// TIA Portal V17 export
// export: Created 2025-03-05T08:01:40.2934801Z, ExportSetting WithDefaults, DisplayName Totally Integrated Automation Portal, DisplayVersion V17 Update 8, DisplayName TIA Portal Openness, DisplayVersion V17 Update 8, DisplayName TIA Portal Version Control Interface, DisplayVersion V17, DisplayName SINAMICS Startdrive Advanced, DisplayVersion V17 SP2, DisplayName SINAMICS Startdrive G110M, G120, G120C, G120D, G120P, G115D, DisplayVersion V17 SP2, DisplayName SINAMICS Startdrive G130, G150, S120, S150, SINAMICS MV, S210, DisplayVersion V17 SP2, DisplayName STEP 7 Professional, DisplayVersion V17 Update 8, DisplayName SINUMERIK ONE STEP 7 Toolbox, DisplayVersion V17 Update 12, DisplayName SINUMERIK 840D sl STEP 7 Toolbox, DisplayVersion V17 Update 12, DisplayName STEP 7 Safety, DisplayVersion V17 Update 6, DisplayName WinCC Advanced, DisplayVersion V17 Update 8
FUNCTION "FC7222_MACHINE_OVERVIEW_CLADDING" : Void   // FC7222, LAD
{ S7_Optimized_Access := 'FALSE' }
AUTHOR : ETXETAR
VERSION : 1.0
// stored: AutoNumber false, IsIECCheckEnabled false, SetENOAutomatically false, UDAEnableTagReadback false
   VAR_TEMP
      OPTION_OFF : Bool;   // OPTION OFF
      OPTION_ON : Bool;   // OPTION ON
      SPINDLE_SP11 : Bool;   // SPINDLE SP11
      SPINDLE_SP12 : Bool;   // SPINDLE SP12
      SPINDLE_SP13 : Bool;   // SPINDLE SP13
      SPINDLE_SP14 : Bool;   // SPINDLE SP14
      SPINDLE_SP21 : Bool;   // SPINDLE SP21
      SPINDLE_SP22 : Bool;   // SPINDLE SP22
      SPINDLE_SP23 : Bool;   // SPINDLE SP23
      SPINDLE_SP24 : Bool;   // SPINDLE SP24
      MACH_FIXTURE_1 : Bool;   // MACH FIXTURE 1
      MACH_FIXTURE_2 : Bool;   // MACH FIXTURE 2
      UNIT_MODE_AUX : Int;   // UNIT MODE AUXILIARY
   END_VAR
   VAR_TEMP   // added for the SCL form of the ladder/FBD networks
      _w1 : Bool;
      _w2 : Bool;
      _w3 : Bool;
      _w4 : Bool;
   END_VAR
BEGIN

REGION Network 1: OPTION OFF
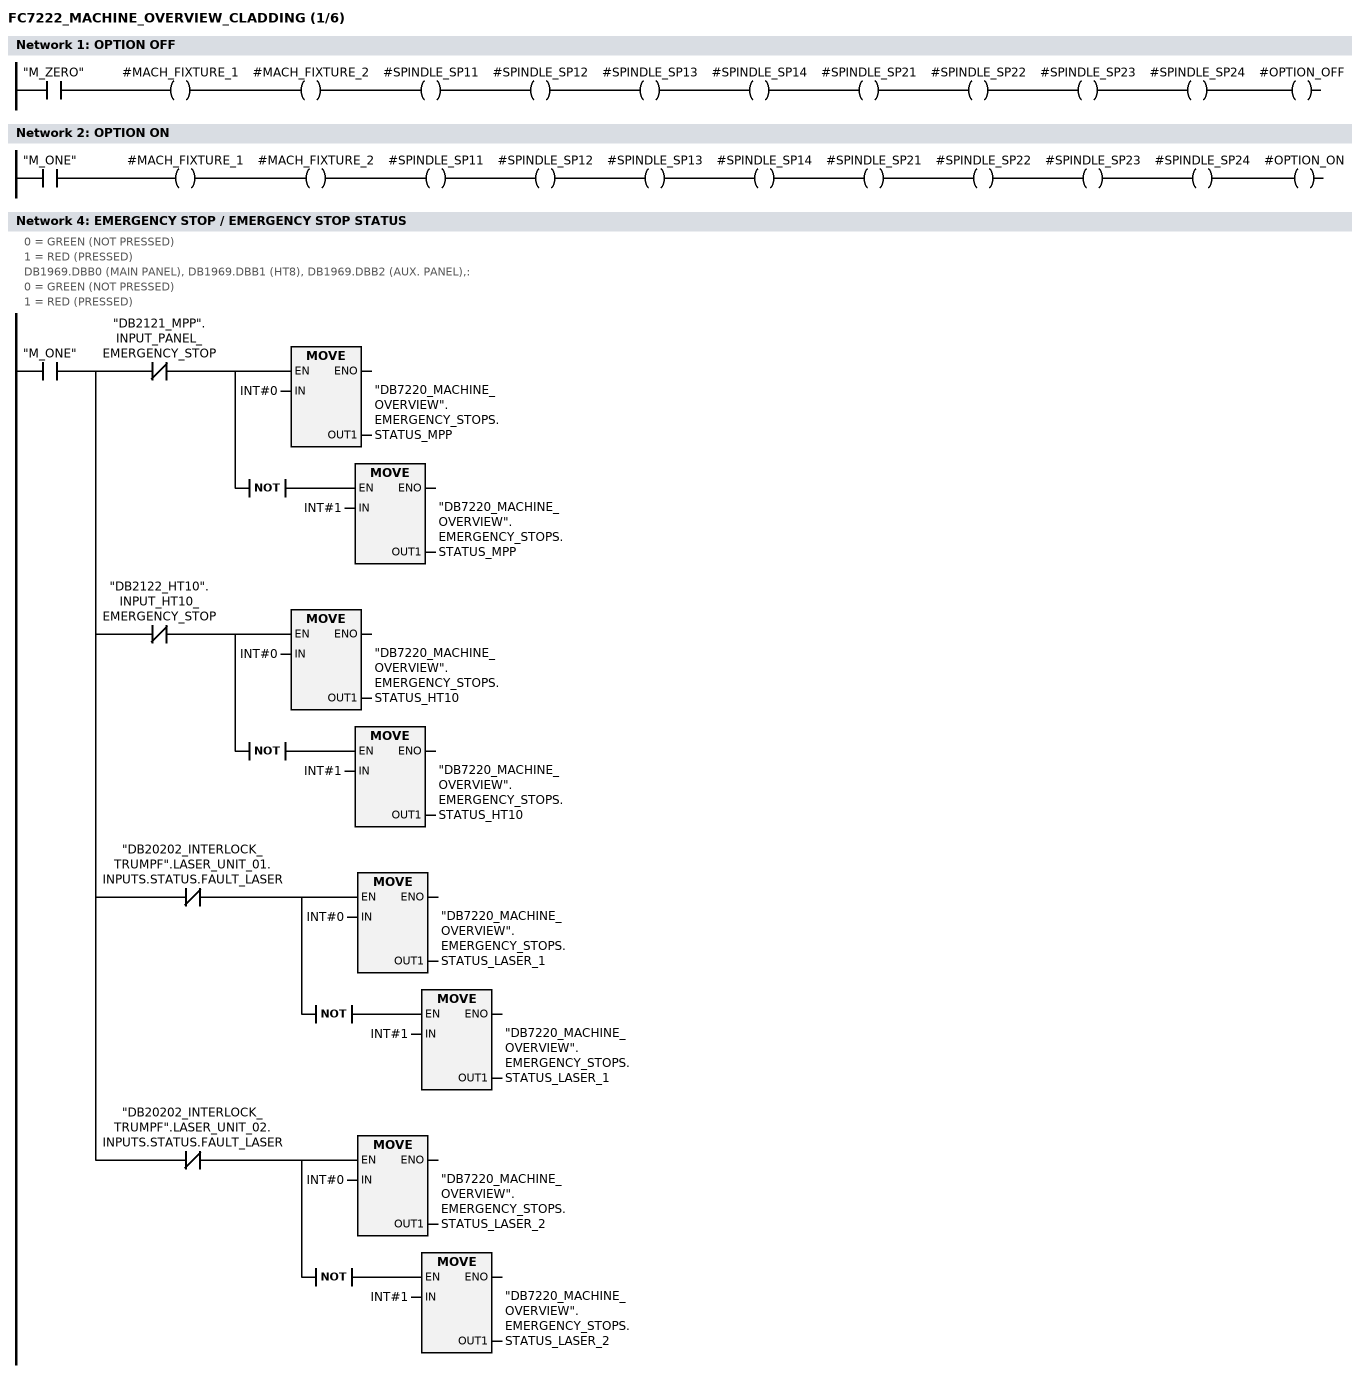
   RUNG wire#powerrail
      Contact( "M_ZERO" )
      Coil( #MACH_FIXTURE_1 )
      Coil( #MACH_FIXTURE_2 )
      Coil( #SPINDLE_SP11 )
      Coil( #SPINDLE_SP12 )
      Coil( #SPINDLE_SP13 )
      Coil( #SPINDLE_SP14 )
      Coil( #SPINDLE_SP21 )
      Coil( #SPINDLE_SP22 )
      Coil( #SPINDLE_SP23 )
      Coil( #SPINDLE_SP24 )
      Coil( #OPTION_OFF )
   END_RUNG
   // the same network as SCL:
   #MACH_FIXTURE_1 := "M_ZERO";
   #MACH_FIXTURE_2 := "M_ZERO";
   #SPINDLE_SP11 := "M_ZERO";
   #SPINDLE_SP12 := "M_ZERO";
   #SPINDLE_SP13 := "M_ZERO";
   #SPINDLE_SP14 := "M_ZERO";
   #SPINDLE_SP21 := "M_ZERO";
   #SPINDLE_SP22 := "M_ZERO";
   #SPINDLE_SP23 := "M_ZERO";
   #SPINDLE_SP24 := "M_ZERO";
   #OPTION_OFF := "M_ZERO";
END_REGION

REGION Network 2: OPTION ON
   RUNG wire#powerrail
      Contact( "M_ONE" )
      Coil( #MACH_FIXTURE_1 )
      Coil( #MACH_FIXTURE_2 )
      Coil( #SPINDLE_SP11 )
      Coil( #SPINDLE_SP12 )
      Coil( #SPINDLE_SP13 )
      Coil( #SPINDLE_SP14 )
      Coil( #SPINDLE_SP21 )
      Coil( #SPINDLE_SP22 )
      Coil( #SPINDLE_SP23 )
      Coil( #SPINDLE_SP24 )
      Coil( #OPTION_ON )
   END_RUNG
   // the same network as SCL:
   #MACH_FIXTURE_1 := "M_ONE";
   #MACH_FIXTURE_2 := "M_ONE";
   #SPINDLE_SP11 := "M_ONE";
   #SPINDLE_SP12 := "M_ONE";
   #SPINDLE_SP13 := "M_ONE";
   #SPINDLE_SP14 := "M_ONE";
   #SPINDLE_SP21 := "M_ONE";
   #SPINDLE_SP22 := "M_ONE";
   #SPINDLE_SP23 := "M_ONE";
   #SPINDLE_SP24 := "M_ONE";
   #OPTION_ON := "M_ONE";
END_REGION

REGION Network 3: ********** EMERGENCY STOP **********
   // MPP PANEL EMERGENCY STOP
   // HT10 EMERGENCY STOP
   // AUXILIAR MAGAZINE PANEL EMERGENCY STOP
   // MANUAL LOADING EMERGENCY STOP
   // CHIP CONVEYOR EMERGENCY STOP
END_REGION

REGION Network 4: EMERGENCY STOP / EMERGENCY STOP STATUS
   // 0 = GREEN (NOT PRESSED)
   // 1 = RED (PRESSED)
   // DB1969.DBB0 (MAIN PANEL), DB1969.DBB1 (HT8), DB1969.DBB2 (AUX. PANEL),:
   // 
   // 0 = GREEN (NOT PRESSED)
   // 
   // 1 = RED (PRESSED)
   RUNG wire#powerrail
      Contact( "M_ONE" )
      wire#w1
      I_Contact( "DB2121_MPP".INPUT_PANEL_EMERGENCY_STOP )
      wire#w2
      { S7_GenerateENO := "TRUE" } Move(in := INT#0, out1 => "DB7220_MACHINE_OVERVIEW".EMERGENCY_STOPS.STATUS_MPP)
   END_RUNG
   RUNG wire#w2
      Not()
      { S7_GenerateENO := "TRUE" } Move(in := INT#1, out1 => "DB7220_MACHINE_OVERVIEW".EMERGENCY_STOPS.STATUS_MPP)
   END_RUNG
   RUNG wire#w1
      I_Contact( "DB2122_HT10".INPUT_HT10_EMERGENCY_STOP )
      wire#w3
      { S7_GenerateENO := "TRUE" } Move(in := INT#0, out1 => "DB7220_MACHINE_OVERVIEW".EMERGENCY_STOPS.STATUS_HT10)
   END_RUNG
   RUNG wire#w3
      Not()
      { S7_GenerateENO := "TRUE" } Move(in := INT#1, out1 => "DB7220_MACHINE_OVERVIEW".EMERGENCY_STOPS.STATUS_HT10)
   END_RUNG
   RUNG wire#w1
      I_Contact( "DB20202_INTERLOCK_TRUMPF".LASER_UNIT_01.INPUTS.STATUS.FAULT_LASER )
      wire#w4
      Move(in := INT#0, out1 => "DB7220_MACHINE_OVERVIEW".EMERGENCY_STOPS.STATUS_LASER_1)
   END_RUNG
   RUNG wire#w4
      Not()
      Move(in := INT#1, out1 => "DB7220_MACHINE_OVERVIEW".EMERGENCY_STOPS.STATUS_LASER_1)
   END_RUNG
   RUNG wire#w1
      I_Contact( "DB20202_INTERLOCK_TRUMPF".LASER_UNIT_02.INPUTS.STATUS.FAULT_LASER )
      wire#w5
      Move(in := INT#0, out1 => "DB7220_MACHINE_OVERVIEW".EMERGENCY_STOPS.STATUS_LASER_2)
   END_RUNG
   RUNG wire#w5
      Not()
      Move(in := INT#1, out1 => "DB7220_MACHINE_OVERVIEW".EMERGENCY_STOPS.STATUS_LASER_2)
   END_RUNG
   // the same network as SCL:
   #_w1 := "M_ONE" AND NOT "DB2121_MPP".INPUT_PANEL_EMERGENCY_STOP;
   IF #_w1 THEN "DB7220_MACHINE_OVERVIEW".EMERGENCY_STOPS.STATUS_MPP := INT#0; END_IF;
   IF NOT #_w1 THEN "DB7220_MACHINE_OVERVIEW".EMERGENCY_STOPS.STATUS_MPP := INT#1; END_IF;
   #_w2 := "M_ONE" AND NOT "DB2122_HT10".INPUT_HT10_EMERGENCY_STOP;
   IF #_w2 THEN "DB7220_MACHINE_OVERVIEW".EMERGENCY_STOPS.STATUS_HT10 := INT#0; END_IF;
   IF NOT #_w2 THEN "DB7220_MACHINE_OVERVIEW".EMERGENCY_STOPS.STATUS_HT10 := INT#1; END_IF;
   #_w3 := "M_ONE" AND NOT "DB20202_INTERLOCK_TRUMPF".LASER_UNIT_01.INPUTS.STATUS.FAULT_LASER;
   IF #_w3 THEN "DB7220_MACHINE_OVERVIEW".EMERGENCY_STOPS.STATUS_LASER_1 := INT#0; END_IF;
   IF NOT #_w3 THEN "DB7220_MACHINE_OVERVIEW".EMERGENCY_STOPS.STATUS_LASER_1 := INT#1; END_IF;
   #_w4 := "M_ONE" AND NOT "DB20202_INTERLOCK_TRUMPF".LASER_UNIT_02.INPUTS.STATUS.FAULT_LASER;
   IF #_w4 THEN "DB7220_MACHINE_OVERVIEW".EMERGENCY_STOPS.STATUS_LASER_2 := INT#0; END_IF;
   IF NOT #_w4 THEN "DB7220_MACHINE_OVERVIEW".EMERGENCY_STOPS.STATUS_LASER_2 := INT#1; END_IF;
END_REGION

REGION Network 5: ********** SAFETY DOORS **********
   // ::::::::::::::::::::::::::::::::::::::::::::::::::::::::::::::::::::::::::::::::
   // :::::::::::::::::::::::::::: SAFETY DOOR STATUS ::::::::::::::::::::::::::::::::
   // ::::::::::::::::::::::::::::::::::::::::::::::::::::::::::::::::::::::::::::::::
   // DELETE THE NETWORKS OF THE DOORS THAT DO NOT EXIST IN THE MACHINE
   // TOOL MAGAZINE 01R SAFETY DOOR
   // TOOL MAGAZINE 01L SAFETY DOOR
   // UNIT 01R SAFETY DOOR
   // UNIT 01L SAFETY DOOR
   // CHIP CONVEYOR SAFETY DOOR
   // AUTOMATIC DOOR
END_REGION

REGION Network 6: UNIT 01 MAIN SAFETY DOOR
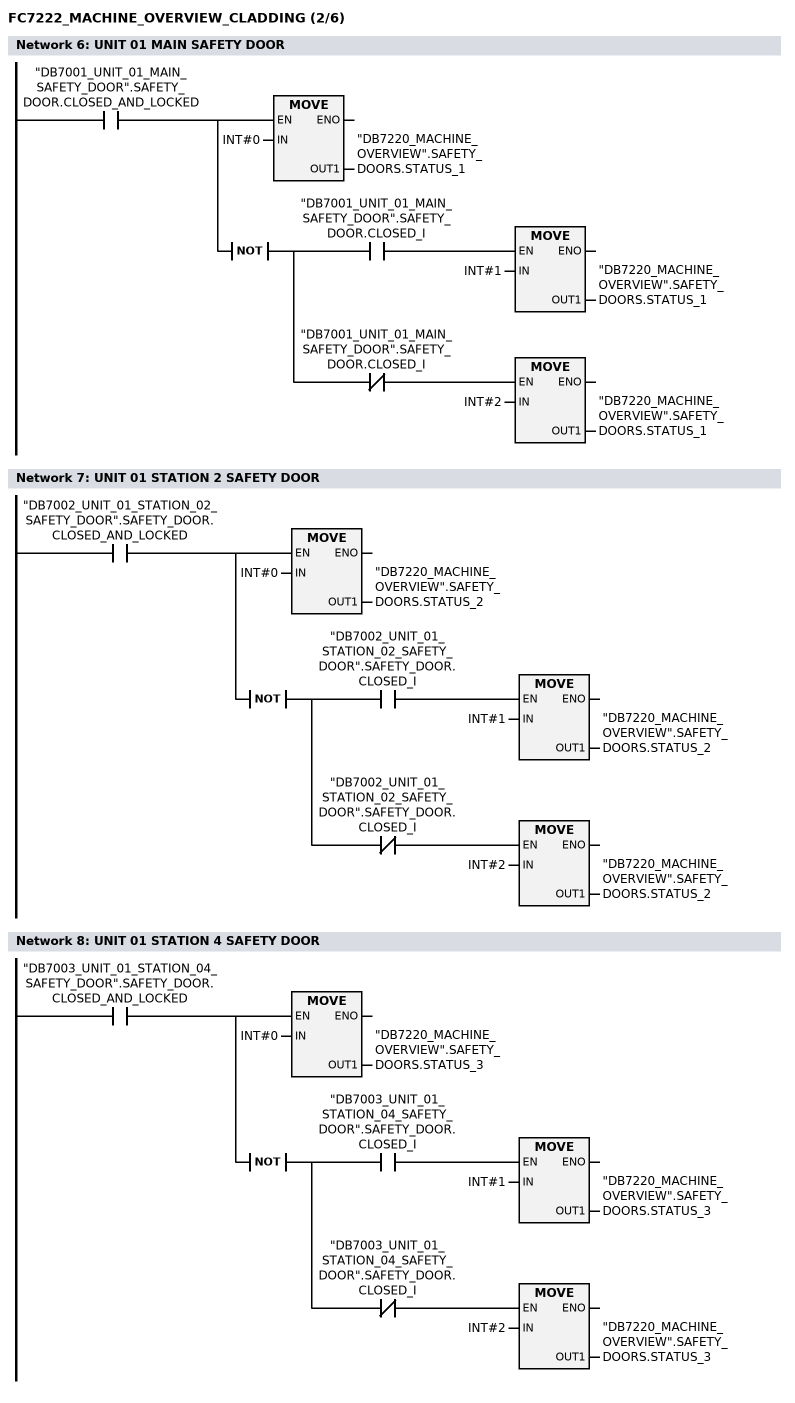
   RUNG wire#powerrail
      Contact( "DB7001_UNIT_01_MAIN_SAFETY_DOOR".SAFETY_DOOR.CLOSED_AND_LOCKED )
      wire#w1
      Move(in := INT#0, out1 => "DB7220_MACHINE_OVERVIEW".SAFETY_DOORS.STATUS_1)
   END_RUNG
   RUNG wire#w1
      Not()
      wire#w2
      Contact( "DB7001_UNIT_01_MAIN_SAFETY_DOOR".SAFETY_DOOR.CLOSED_I )
      Move(in := INT#1, out1 => "DB7220_MACHINE_OVERVIEW".SAFETY_DOORS.STATUS_1)
   END_RUNG
   RUNG wire#w2
      I_Contact( "DB7001_UNIT_01_MAIN_SAFETY_DOOR".SAFETY_DOOR.CLOSED_I )
      Move(in := INT#2, out1 => "DB7220_MACHINE_OVERVIEW".SAFETY_DOORS.STATUS_1)
   END_RUNG
   // the same network as SCL:
   IF "DB7001_UNIT_01_MAIN_SAFETY_DOOR".SAFETY_DOOR.CLOSED_AND_LOCKED THEN
       "DB7220_MACHINE_OVERVIEW".SAFETY_DOORS.STATUS_1 := INT#0;
   END_IF;
   #_w1 := NOT "DB7001_UNIT_01_MAIN_SAFETY_DOOR".SAFETY_DOOR.CLOSED_AND_LOCKED;
   IF #_w1 AND "DB7001_UNIT_01_MAIN_SAFETY_DOOR".SAFETY_DOOR.CLOSED_I THEN
       "DB7220_MACHINE_OVERVIEW".SAFETY_DOORS.STATUS_1 := INT#1;
   END_IF;
   IF #_w1 AND NOT "DB7001_UNIT_01_MAIN_SAFETY_DOOR".SAFETY_DOOR.CLOSED_I THEN
       "DB7220_MACHINE_OVERVIEW".SAFETY_DOORS.STATUS_1 := INT#2;
   END_IF;
END_REGION

REGION Network 7: UNIT 01 STATION 2 SAFETY DOOR
   RUNG wire#powerrail
      Contact( "DB7002_UNIT_01_STATION_02_SAFETY_DOOR".SAFETY_DOOR.CLOSED_AND_LOCKED )
      wire#w1
      Move(in := INT#0, out1 => "DB7220_MACHINE_OVERVIEW".SAFETY_DOORS.STATUS_2)
   END_RUNG
   RUNG wire#w1
      Not()
      wire#w2
      Contact( "DB7002_UNIT_01_STATION_02_SAFETY_DOOR".SAFETY_DOOR.CLOSED_I )
      Move(in := INT#1, out1 => "DB7220_MACHINE_OVERVIEW".SAFETY_DOORS.STATUS_2)
   END_RUNG
   RUNG wire#w2
      I_Contact( "DB7002_UNIT_01_STATION_02_SAFETY_DOOR".SAFETY_DOOR.CLOSED_I )
      Move(in := INT#2, out1 => "DB7220_MACHINE_OVERVIEW".SAFETY_DOORS.STATUS_2)
   END_RUNG
   // the same network as SCL:
   IF "DB7002_UNIT_01_STATION_02_SAFETY_DOOR".SAFETY_DOOR.CLOSED_AND_LOCKED THEN
       "DB7220_MACHINE_OVERVIEW".SAFETY_DOORS.STATUS_2 := INT#0;
   END_IF;
   #_w1 := NOT "DB7002_UNIT_01_STATION_02_SAFETY_DOOR".SAFETY_DOOR.CLOSED_AND_LOCKED;
   IF #_w1 AND "DB7002_UNIT_01_STATION_02_SAFETY_DOOR".SAFETY_DOOR.CLOSED_I THEN
       "DB7220_MACHINE_OVERVIEW".SAFETY_DOORS.STATUS_2 := INT#1;
   END_IF;
   IF #_w1 AND NOT "DB7002_UNIT_01_STATION_02_SAFETY_DOOR".SAFETY_DOOR.CLOSED_I THEN
       "DB7220_MACHINE_OVERVIEW".SAFETY_DOORS.STATUS_2 := INT#2;
   END_IF;
END_REGION

REGION Network 8: UNIT 01 STATION 4 SAFETY DOOR
   RUNG wire#powerrail
      Contact( "DB7003_UNIT_01_STATION_04_SAFETY_DOOR".SAFETY_DOOR.CLOSED_AND_LOCKED )
      wire#w1
      Move(in := INT#0, out1 => "DB7220_MACHINE_OVERVIEW".SAFETY_DOORS.STATUS_3)
   END_RUNG
   RUNG wire#w1
      Not()
      wire#w2
      Contact( "DB7003_UNIT_01_STATION_04_SAFETY_DOOR".SAFETY_DOOR.CLOSED_I )
      Move(in := INT#1, out1 => "DB7220_MACHINE_OVERVIEW".SAFETY_DOORS.STATUS_3)
   END_RUNG
   RUNG wire#w2
      I_Contact( "DB7003_UNIT_01_STATION_04_SAFETY_DOOR".SAFETY_DOOR.CLOSED_I )
      Move(in := INT#2, out1 => "DB7220_MACHINE_OVERVIEW".SAFETY_DOORS.STATUS_3)
   END_RUNG
   // the same network as SCL:
   IF "DB7003_UNIT_01_STATION_04_SAFETY_DOOR".SAFETY_DOOR.CLOSED_AND_LOCKED THEN
       "DB7220_MACHINE_OVERVIEW".SAFETY_DOORS.STATUS_3 := INT#0;
   END_IF;
   #_w1 := NOT "DB7003_UNIT_01_STATION_04_SAFETY_DOOR".SAFETY_DOOR.CLOSED_AND_LOCKED;
   IF #_w1 AND "DB7003_UNIT_01_STATION_04_SAFETY_DOOR".SAFETY_DOOR.CLOSED_I THEN
       "DB7220_MACHINE_OVERVIEW".SAFETY_DOORS.STATUS_3 := INT#1;
   END_IF;
   IF #_w1 AND NOT "DB7003_UNIT_01_STATION_04_SAFETY_DOOR".SAFETY_DOOR.CLOSED_I THEN
       "DB7220_MACHINE_OVERVIEW".SAFETY_DOORS.STATUS_3 := INT#2;
   END_IF;
END_REGION

REGION Network 9: UNIT 02 MAIN SAFETY DOOR
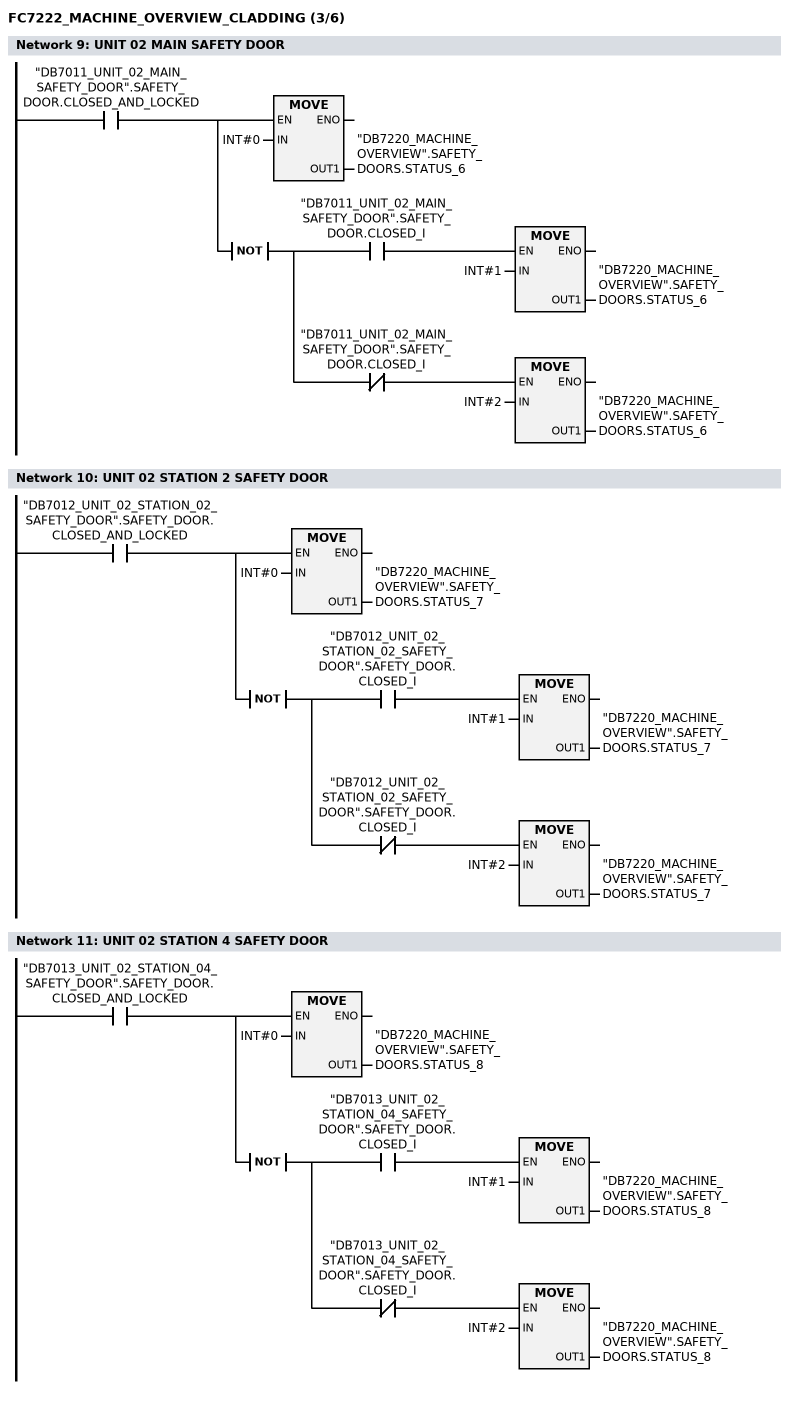
   RUNG wire#powerrail
      Contact( "DB7011_UNIT_02_MAIN_SAFETY_DOOR".SAFETY_DOOR.CLOSED_AND_LOCKED )
      wire#w1
      Move(in := INT#0, out1 => "DB7220_MACHINE_OVERVIEW".SAFETY_DOORS.STATUS_6)
   END_RUNG
   RUNG wire#w1
      Not()
      wire#w2
      Contact( "DB7011_UNIT_02_MAIN_SAFETY_DOOR".SAFETY_DOOR.CLOSED_I )
      Move(in := INT#1, out1 => "DB7220_MACHINE_OVERVIEW".SAFETY_DOORS.STATUS_6)
   END_RUNG
   RUNG wire#w2
      I_Contact( "DB7011_UNIT_02_MAIN_SAFETY_DOOR".SAFETY_DOOR.CLOSED_I )
      Move(in := INT#2, out1 => "DB7220_MACHINE_OVERVIEW".SAFETY_DOORS.STATUS_6)
   END_RUNG
   // the same network as SCL:
   IF "DB7011_UNIT_02_MAIN_SAFETY_DOOR".SAFETY_DOOR.CLOSED_AND_LOCKED THEN
       "DB7220_MACHINE_OVERVIEW".SAFETY_DOORS.STATUS_6 := INT#0;
   END_IF;
   #_w1 := NOT "DB7011_UNIT_02_MAIN_SAFETY_DOOR".SAFETY_DOOR.CLOSED_AND_LOCKED;
   IF #_w1 AND "DB7011_UNIT_02_MAIN_SAFETY_DOOR".SAFETY_DOOR.CLOSED_I THEN
       "DB7220_MACHINE_OVERVIEW".SAFETY_DOORS.STATUS_6 := INT#1;
   END_IF;
   IF #_w1 AND NOT "DB7011_UNIT_02_MAIN_SAFETY_DOOR".SAFETY_DOOR.CLOSED_I THEN
       "DB7220_MACHINE_OVERVIEW".SAFETY_DOORS.STATUS_6 := INT#2;
   END_IF;
END_REGION

REGION Network 10: UNIT 02 STATION 2 SAFETY DOOR
   RUNG wire#powerrail
      Contact( "DB7012_UNIT_02_STATION_02_SAFETY_DOOR".SAFETY_DOOR.CLOSED_AND_LOCKED )
      wire#w1
      Move(in := INT#0, out1 => "DB7220_MACHINE_OVERVIEW".SAFETY_DOORS.STATUS_7)
   END_RUNG
   RUNG wire#w1
      Not()
      wire#w2
      Contact( "DB7012_UNIT_02_STATION_02_SAFETY_DOOR".SAFETY_DOOR.CLOSED_I )
      Move(in := INT#1, out1 => "DB7220_MACHINE_OVERVIEW".SAFETY_DOORS.STATUS_7)
   END_RUNG
   RUNG wire#w2
      I_Contact( "DB7012_UNIT_02_STATION_02_SAFETY_DOOR".SAFETY_DOOR.CLOSED_I )
      Move(in := INT#2, out1 => "DB7220_MACHINE_OVERVIEW".SAFETY_DOORS.STATUS_7)
   END_RUNG
   // the same network as SCL:
   IF "DB7012_UNIT_02_STATION_02_SAFETY_DOOR".SAFETY_DOOR.CLOSED_AND_LOCKED THEN
       "DB7220_MACHINE_OVERVIEW".SAFETY_DOORS.STATUS_7 := INT#0;
   END_IF;
   #_w1 := NOT "DB7012_UNIT_02_STATION_02_SAFETY_DOOR".SAFETY_DOOR.CLOSED_AND_LOCKED;
   IF #_w1 AND "DB7012_UNIT_02_STATION_02_SAFETY_DOOR".SAFETY_DOOR.CLOSED_I THEN
       "DB7220_MACHINE_OVERVIEW".SAFETY_DOORS.STATUS_7 := INT#1;
   END_IF;
   IF #_w1 AND NOT "DB7012_UNIT_02_STATION_02_SAFETY_DOOR".SAFETY_DOOR.CLOSED_I THEN
       "DB7220_MACHINE_OVERVIEW".SAFETY_DOORS.STATUS_7 := INT#2;
   END_IF;
END_REGION

REGION Network 11: UNIT 02 STATION 4 SAFETY DOOR
   RUNG wire#powerrail
      Contact( "DB7013_UNIT_02_STATION_04_SAFETY_DOOR".SAFETY_DOOR.CLOSED_AND_LOCKED )
      wire#w1
      Move(in := INT#0, out1 => "DB7220_MACHINE_OVERVIEW".SAFETY_DOORS.STATUS_8)
   END_RUNG
   RUNG wire#w1
      Not()
      wire#w2
      Contact( "DB7013_UNIT_02_STATION_04_SAFETY_DOOR".SAFETY_DOOR.CLOSED_I )
      Move(in := INT#1, out1 => "DB7220_MACHINE_OVERVIEW".SAFETY_DOORS.STATUS_8)
   END_RUNG
   RUNG wire#w2
      I_Contact( "DB7013_UNIT_02_STATION_04_SAFETY_DOOR".SAFETY_DOOR.CLOSED_I )
      Move(in := INT#2, out1 => "DB7220_MACHINE_OVERVIEW".SAFETY_DOORS.STATUS_8)
   END_RUNG
   // the same network as SCL:
   IF "DB7013_UNIT_02_STATION_04_SAFETY_DOOR".SAFETY_DOOR.CLOSED_AND_LOCKED THEN
       "DB7220_MACHINE_OVERVIEW".SAFETY_DOORS.STATUS_8 := INT#0;
   END_IF;
   #_w1 := NOT "DB7013_UNIT_02_STATION_04_SAFETY_DOOR".SAFETY_DOOR.CLOSED_AND_LOCKED;
   IF #_w1 AND "DB7013_UNIT_02_STATION_04_SAFETY_DOOR".SAFETY_DOOR.CLOSED_I THEN
       "DB7220_MACHINE_OVERVIEW".SAFETY_DOORS.STATUS_8 := INT#1;
   END_IF;
   IF #_w1 AND NOT "DB7013_UNIT_02_STATION_04_SAFETY_DOOR".SAFETY_DOOR.CLOSED_I THEN
       "DB7220_MACHINE_OVERVIEW".SAFETY_DOORS.STATUS_8 := INT#2;
   END_IF;
END_REGION

REGION Network 12: ********** UNITS **********
END_REGION

REGION Network 13: UNIT MODE STATUS
   // 0 = GREEN (AUTO)
   // 
   // 1 = BLUE (MANUAL)
   // 
   // 2 = YELLOW (MDA) 
   // 
   // 3 = WHITE (SEMIAUTOMATIC)
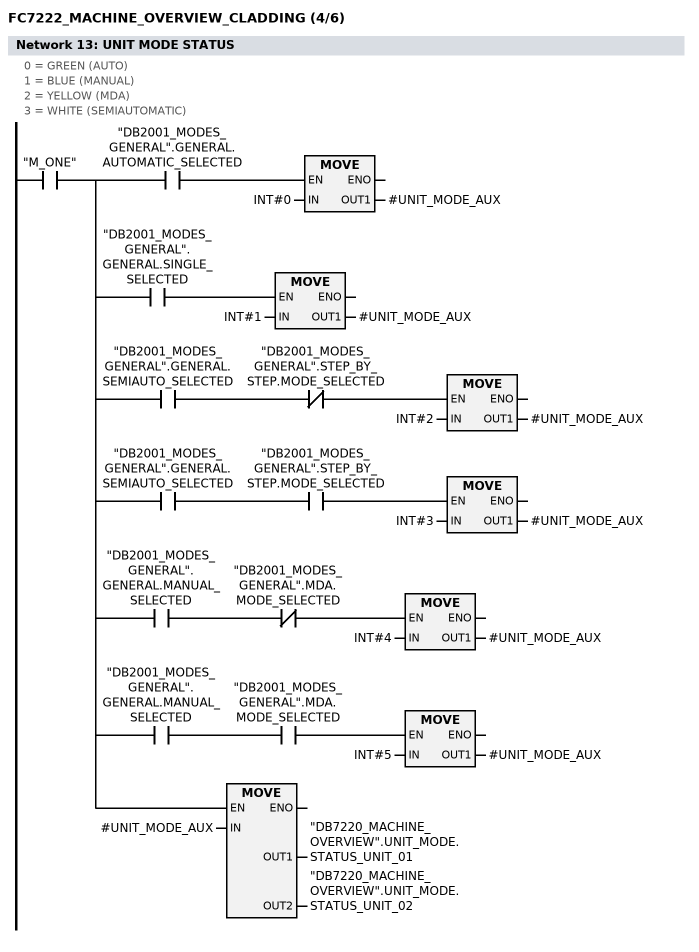
   RUNG wire#powerrail
      Contact( "M_ONE" )
      wire#w1
      Contact( "DB2001_MODES_GENERAL".GENERAL.AUTOMATIC_SELECTED )
      { S7_GenerateENO := "TRUE" } Move(in := INT#0, out1 => #UNIT_MODE_AUX)
   END_RUNG
   RUNG wire#w1
      Contact( "DB2001_MODES_GENERAL".GENERAL.SINGLE_SELECTED )
      { S7_GenerateENO := "TRUE" } Move(in := INT#1, out1 => #UNIT_MODE_AUX)
   END_RUNG
   RUNG wire#w1
      Contact( "DB2001_MODES_GENERAL".GENERAL.SEMIAUTO_SELECTED )
      I_Contact( "DB2001_MODES_GENERAL".STEP_BY_STEP.MODE_SELECTED )
      { S7_GenerateENO := "TRUE" } Move(in := INT#2, out1 => #UNIT_MODE_AUX)
   END_RUNG
   RUNG wire#w1
      Contact( "DB2001_MODES_GENERAL".GENERAL.SEMIAUTO_SELECTED )
      Contact( "DB2001_MODES_GENERAL".STEP_BY_STEP.MODE_SELECTED )
      { S7_GenerateENO := "TRUE" } Move(in := INT#3, out1 => #UNIT_MODE_AUX)
   END_RUNG
   RUNG wire#w1
      Contact( "DB2001_MODES_GENERAL".GENERAL.MANUAL_SELECTED )
      I_Contact( "DB2001_MODES_GENERAL".MDA.MODE_SELECTED )
      { S7_GenerateENO := "TRUE" } Move(in := INT#4, out1 => #UNIT_MODE_AUX)
   END_RUNG
   RUNG wire#w1
      Contact( "DB2001_MODES_GENERAL".GENERAL.MANUAL_SELECTED )
      Contact( "DB2001_MODES_GENERAL".MDA.MODE_SELECTED )
      { S7_GenerateENO := "TRUE" } Move(in := INT#5, out1 => #UNIT_MODE_AUX)
   END_RUNG
   RUNG wire#w1
      { S7_GenerateENO := "TRUE" } Move(in := #UNIT_MODE_AUX, out1 => "DB7220_MACHINE_OVERVIEW".UNIT_MODE.STATUS_UNIT_01, out2 => "DB7220_MACHINE_OVERVIEW".UNIT_MODE.STATUS_UNIT_02)
   END_RUNG
   // the same network as SCL:
   IF "M_ONE" AND "DB2001_MODES_GENERAL".GENERAL.AUTOMATIC_SELECTED THEN #UNIT_MODE_AUX := INT#0; END_IF;
   IF "M_ONE" AND "DB2001_MODES_GENERAL".GENERAL.SINGLE_SELECTED THEN #UNIT_MODE_AUX := INT#1; END_IF;
   IF "M_ONE" AND "DB2001_MODES_GENERAL".GENERAL.SEMIAUTO_SELECTED AND NOT "DB2001_MODES_GENERAL".STEP_BY_STEP.MODE_SELECTED THEN
       #UNIT_MODE_AUX := INT#2;
   END_IF;
   IF "M_ONE" AND "DB2001_MODES_GENERAL".GENERAL.SEMIAUTO_SELECTED AND "DB2001_MODES_GENERAL".STEP_BY_STEP.MODE_SELECTED THEN
       #UNIT_MODE_AUX := INT#3;
   END_IF;
   IF "M_ONE" AND "DB2001_MODES_GENERAL".GENERAL.MANUAL_SELECTED AND NOT "DB2001_MODES_GENERAL".MDA.MODE_SELECTED THEN
       #UNIT_MODE_AUX := INT#4;
   END_IF;
   IF "M_ONE" AND "DB2001_MODES_GENERAL".GENERAL.MANUAL_SELECTED AND "DB2001_MODES_GENERAL".MDA.MODE_SELECTED THEN
       #UNIT_MODE_AUX := INT#5;
   END_IF;
   IF "M_ONE" THEN
       "DB7220_MACHINE_OVERVIEW".UNIT_MODE.STATUS_UNIT_01 := #UNIT_MODE_AUX;
       "DB7220_MACHINE_OVERVIEW".UNIT_MODE.STATUS_UNIT_02 := #UNIT_MODE_AUX;
   END_IF;
END_REGION

REGION Network 14: UNITS STATUS / MACHINE STATUS UNIT 01R FIELD (UNIT)
   // 0 = GREEN (CYCLE ON)
   // 
   // 1 = YELLOW (WARNING)
   // 
   // 2 = RED    (ALARM)
   // DB1969.DBB60: UNIT 01R
   // 
   // 0 = GREEN (CYCLE ON)
   // 
   // 1 = YELLOW (WARNING)
   // 
   // 2 = RED    (ALARM)
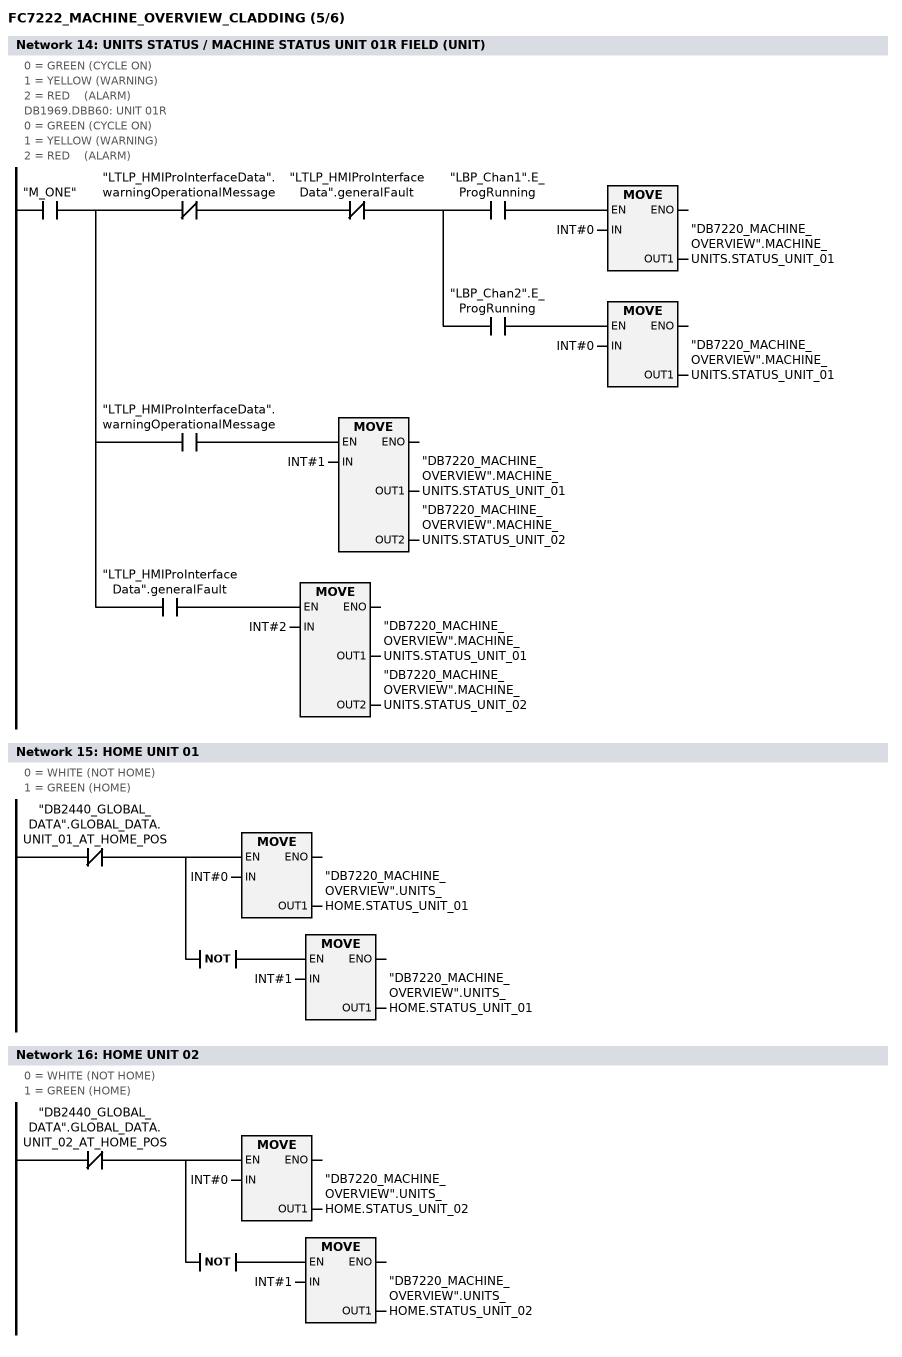
   RUNG wire#powerrail
      Contact( "M_ONE" )
      wire#w1
      I_Contact( "LTLP_HMIProInterfaceData".warningOperationalMessage )
      I_Contact( "LTLP_HMIProInterfaceData".generalFault )
      wire#w2
      Contact( "LBP_Chan1".E_ProgRunning )
      { S7_GenerateENO := "TRUE" } Move(in := INT#0, out1 => "DB7220_MACHINE_OVERVIEW".MACHINE_UNITS.STATUS_UNIT_01)
   END_RUNG
   RUNG wire#w2
      Contact( "LBP_Chan2".E_ProgRunning )
      { S7_GenerateENO := "TRUE" } Move(in := INT#0, out1 => "DB7220_MACHINE_OVERVIEW".MACHINE_UNITS.STATUS_UNIT_01)
   END_RUNG
   RUNG wire#w1
      Contact( "LTLP_HMIProInterfaceData".warningOperationalMessage )
      { S7_GenerateENO := "TRUE" } Move(in := INT#1, out1 => "DB7220_MACHINE_OVERVIEW".MACHINE_UNITS.STATUS_UNIT_01, out2 => "DB7220_MACHINE_OVERVIEW".MACHINE_UNITS.STATUS_UNIT_02)
   END_RUNG
   RUNG wire#w1
      Contact( "LTLP_HMIProInterfaceData".generalFault )
      { S7_GenerateENO := "TRUE" } Move(in := INT#2, out1 => "DB7220_MACHINE_OVERVIEW".MACHINE_UNITS.STATUS_UNIT_01, out2 => "DB7220_MACHINE_OVERVIEW".MACHINE_UNITS.STATUS_UNIT_02)
   END_RUNG
   // the same network as SCL:
   #_w1 := "M_ONE" AND NOT "LTLP_HMIProInterfaceData".warningOperationalMessage AND NOT "LTLP_HMIProInterfaceData".generalFault;
   IF #_w1 AND "LBP_Chan1".E_ProgRunning THEN
       "DB7220_MACHINE_OVERVIEW".MACHINE_UNITS.STATUS_UNIT_01 := INT#0;
   END_IF;
   IF #_w1 AND "LBP_Chan2".E_ProgRunning THEN
       "DB7220_MACHINE_OVERVIEW".MACHINE_UNITS.STATUS_UNIT_01 := INT#0;
   END_IF;
   IF "M_ONE" AND "LTLP_HMIProInterfaceData".warningOperationalMessage THEN
       "DB7220_MACHINE_OVERVIEW".MACHINE_UNITS.STATUS_UNIT_01 := INT#1;
       "DB7220_MACHINE_OVERVIEW".MACHINE_UNITS.STATUS_UNIT_02 := INT#1;
   END_IF;
   IF "M_ONE" AND "LTLP_HMIProInterfaceData".generalFault THEN
       "DB7220_MACHINE_OVERVIEW".MACHINE_UNITS.STATUS_UNIT_01 := INT#2;
       "DB7220_MACHINE_OVERVIEW".MACHINE_UNITS.STATUS_UNIT_02 := INT#2;
   END_IF;
END_REGION

REGION Network 15: HOME UNIT 01
   // 0 = WHITE (NOT HOME)
   // 
   // 1 = GREEN (HOME)
   RUNG wire#powerrail
      I_Contact( "DB2440_GLOBAL_DATA".GLOBAL_DATA.UNIT_01_AT_HOME_POS )
      wire#w1
      { S7_GenerateENO := "TRUE" } Move(in := INT#0, out1 => "DB7220_MACHINE_OVERVIEW".UNITS_HOME.STATUS_UNIT_01)
   END_RUNG
   RUNG wire#w1
      Not()
      { S7_GenerateENO := "TRUE" } Move(in := INT#1, out1 => "DB7220_MACHINE_OVERVIEW".UNITS_HOME.STATUS_UNIT_01)
   END_RUNG
   // the same network as SCL:
   #_w1 := NOT "DB2440_GLOBAL_DATA".GLOBAL_DATA.UNIT_01_AT_HOME_POS;
   IF #_w1 THEN "DB7220_MACHINE_OVERVIEW".UNITS_HOME.STATUS_UNIT_01 := INT#0; END_IF;
   IF NOT #_w1 THEN "DB7220_MACHINE_OVERVIEW".UNITS_HOME.STATUS_UNIT_01 := INT#1; END_IF;
END_REGION

REGION Network 16: HOME UNIT 02
   // 0 = WHITE (NOT HOME)
   // 
   // 1 = GREEN (HOME)
   RUNG wire#powerrail
      I_Contact( "DB2440_GLOBAL_DATA".GLOBAL_DATA.UNIT_02_AT_HOME_POS )
      wire#w1
      { S7_GenerateENO := "TRUE" } Move(in := INT#0, out1 => "DB7220_MACHINE_OVERVIEW".UNITS_HOME.STATUS_UNIT_02)
   END_RUNG
   RUNG wire#w1
      Not()
      { S7_GenerateENO := "TRUE" } Move(in := INT#1, out1 => "DB7220_MACHINE_OVERVIEW".UNITS_HOME.STATUS_UNIT_02)
   END_RUNG
   // the same network as SCL:
   #_w1 := NOT "DB2440_GLOBAL_DATA".GLOBAL_DATA.UNIT_02_AT_HOME_POS;
   IF #_w1 THEN "DB7220_MACHINE_OVERVIEW".UNITS_HOME.STATUS_UNIT_02 := INT#0; END_IF;
   IF NOT #_w1 THEN "DB7220_MACHINE_OVERVIEW".UNITS_HOME.STATUS_UNIT_02 := INT#1; END_IF;
END_REGION

REGION Network 17: ********** FIXTURE 1 **********
END_REGION

REGION Network 18: FULL DEPTHS
   // 0 = WHITE (NOT DONE)
   // 
   // 1 = BLUE (DONE)
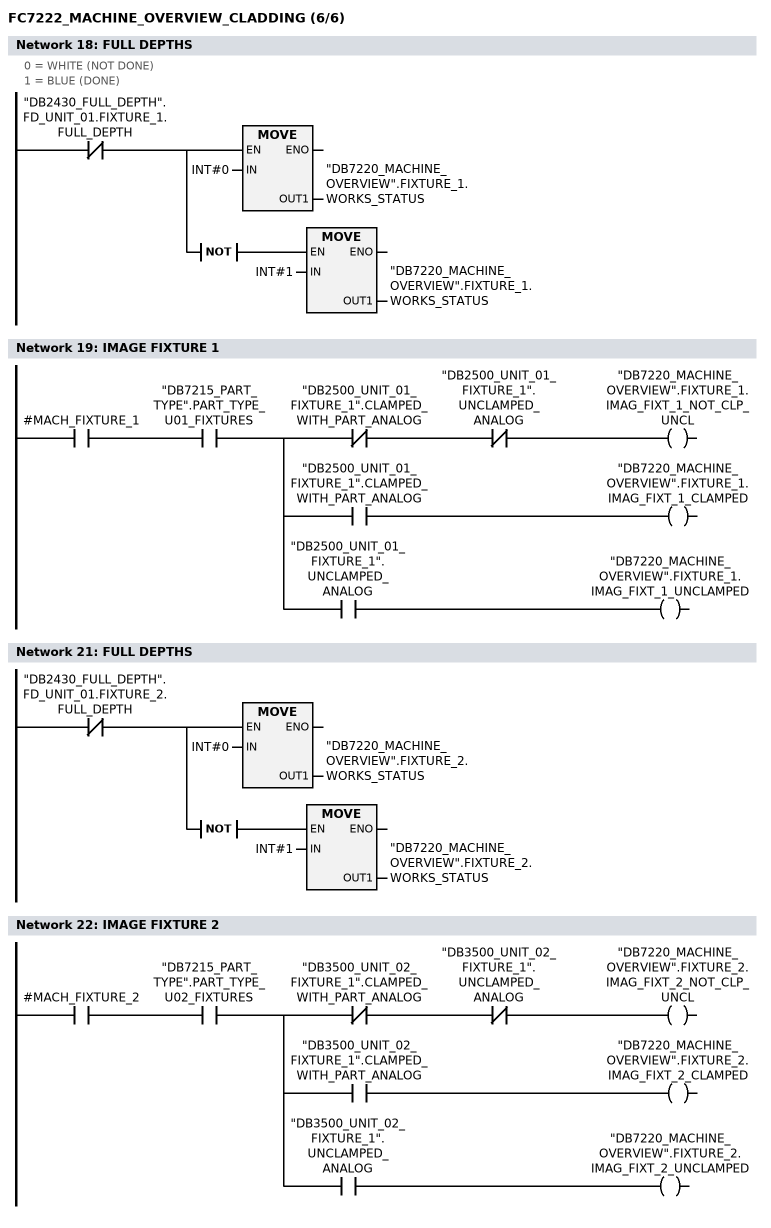
   RUNG wire#powerrail
      I_Contact( "DB2430_FULL_DEPTH".FD_UNIT_01.FIXTURE_1.FULL_DEPTH )
      wire#w1
      { S7_GenerateENO := "TRUE" } Move(in := INT#0, out1 => "DB7220_MACHINE_OVERVIEW".FIXTURE_1.WORKS_STATUS)
   END_RUNG
   RUNG wire#w1
      Not()
      { S7_GenerateENO := "TRUE" } Move(in := INT#1, out1 => "DB7220_MACHINE_OVERVIEW".FIXTURE_1.WORKS_STATUS)
   END_RUNG
   // the same network as SCL:
   #_w1 := NOT "DB2430_FULL_DEPTH".FD_UNIT_01.FIXTURE_1.FULL_DEPTH;
   IF #_w1 THEN "DB7220_MACHINE_OVERVIEW".FIXTURE_1.WORKS_STATUS := INT#0; END_IF;
   IF NOT #_w1 THEN "DB7220_MACHINE_OVERVIEW".FIXTURE_1.WORKS_STATUS := INT#1; END_IF;
END_REGION

REGION Network 19: IMAGE FIXTURE 1
   RUNG wire#powerrail
      Contact( #MACH_FIXTURE_1 )
      Contact( "DB7215_PART_TYPE".PART_TYPE_U01_FIXTURES )
      wire#w1
      I_Contact( "DB2500_UNIT_01_FIXTURE_1".CLAMPED_WITH_PART_ANALOG )
      I_Contact( "DB2500_UNIT_01_FIXTURE_1".UNCLAMPED_ANALOG )
      Coil( "DB7220_MACHINE_OVERVIEW".FIXTURE_1.IMAG_FIXT_1_NOT_CLP_UNCL )
   END_RUNG
   RUNG wire#w1
      Contact( "DB2500_UNIT_01_FIXTURE_1".CLAMPED_WITH_PART_ANALOG )
      Coil( "DB7220_MACHINE_OVERVIEW".FIXTURE_1.IMAG_FIXT_1_CLAMPED )
   END_RUNG
   RUNG wire#w1
      Contact( "DB2500_UNIT_01_FIXTURE_1".UNCLAMPED_ANALOG )
      Coil( "DB7220_MACHINE_OVERVIEW".FIXTURE_1.IMAG_FIXT_1_UNCLAMPED )
   END_RUNG
   // the same network as SCL:
   #_w1 := #MACH_FIXTURE_1 AND "DB7215_PART_TYPE".PART_TYPE_U01_FIXTURES;
   "DB7220_MACHINE_OVERVIEW".FIXTURE_1.IMAG_FIXT_1_NOT_CLP_UNCL := #_w1 AND NOT "DB2500_UNIT_01_FIXTURE_1".CLAMPED_WITH_PART_ANALOG AND NOT "DB2500_UNIT_01_FIXTURE_1".UNCLAMPED_ANALOG;
   "DB7220_MACHINE_OVERVIEW".FIXTURE_1.IMAG_FIXT_1_CLAMPED := #_w1 AND "DB2500_UNIT_01_FIXTURE_1".CLAMPED_WITH_PART_ANALOG;
   "DB7220_MACHINE_OVERVIEW".FIXTURE_1.IMAG_FIXT_1_UNCLAMPED := #_w1 AND "DB2500_UNIT_01_FIXTURE_1".UNCLAMPED_ANALOG;
END_REGION

REGION Network 20: ********** FIXTURE 2 **********
END_REGION

REGION Network 21: FULL DEPTHS
   RUNG wire#powerrail
      I_Contact( "DB2430_FULL_DEPTH".FD_UNIT_01.FIXTURE_2.FULL_DEPTH )
      wire#w1
      { S7_GenerateENO := "TRUE" } Move(in := INT#0, out1 => "DB7220_MACHINE_OVERVIEW".FIXTURE_2.WORKS_STATUS)
   END_RUNG
   RUNG wire#w1
      Not()
      { S7_GenerateENO := "TRUE" } Move(in := INT#1, out1 => "DB7220_MACHINE_OVERVIEW".FIXTURE_2.WORKS_STATUS)
   END_RUNG
   // the same network as SCL:
   #_w1 := NOT "DB2430_FULL_DEPTH".FD_UNIT_01.FIXTURE_2.FULL_DEPTH;
   IF #_w1 THEN "DB7220_MACHINE_OVERVIEW".FIXTURE_2.WORKS_STATUS := INT#0; END_IF;
   IF NOT #_w1 THEN "DB7220_MACHINE_OVERVIEW".FIXTURE_2.WORKS_STATUS := INT#1; END_IF;
END_REGION

REGION Network 22: IMAGE FIXTURE 2
   RUNG wire#powerrail
      Contact( #MACH_FIXTURE_2 )
      Contact( "DB7215_PART_TYPE".PART_TYPE_U02_FIXTURES )
      wire#w1
      I_Contact( "DB3500_UNIT_02_FIXTURE_1".CLAMPED_WITH_PART_ANALOG )
      I_Contact( "DB3500_UNIT_02_FIXTURE_1".UNCLAMPED_ANALOG )
      Coil( "DB7220_MACHINE_OVERVIEW".FIXTURE_2.IMAG_FIXT_2_NOT_CLP_UNCL )
   END_RUNG
   RUNG wire#w1
      Contact( "DB3500_UNIT_02_FIXTURE_1".CLAMPED_WITH_PART_ANALOG )
      Coil( "DB7220_MACHINE_OVERVIEW".FIXTURE_2.IMAG_FIXT_2_CLAMPED )
   END_RUNG
   RUNG wire#w1
      Contact( "DB3500_UNIT_02_FIXTURE_1".UNCLAMPED_ANALOG )
      Coil( "DB7220_MACHINE_OVERVIEW".FIXTURE_2.IMAG_FIXT_2_UNCLAMPED )
   END_RUNG
   // the same network as SCL:
   #_w1 := #MACH_FIXTURE_2 AND "DB7215_PART_TYPE".PART_TYPE_U02_FIXTURES;
   "DB7220_MACHINE_OVERVIEW".FIXTURE_2.IMAG_FIXT_2_NOT_CLP_UNCL := #_w1 AND NOT "DB3500_UNIT_02_FIXTURE_1".CLAMPED_WITH_PART_ANALOG AND NOT "DB3500_UNIT_02_FIXTURE_1".UNCLAMPED_ANALOG;
   "DB7220_MACHINE_OVERVIEW".FIXTURE_2.IMAG_FIXT_2_CLAMPED := #_w1 AND "DB3500_UNIT_02_FIXTURE_1".CLAMPED_WITH_PART_ANALOG;
   "DB7220_MACHINE_OVERVIEW".FIXTURE_2.IMAG_FIXT_2_UNCLAMPED := #_w1 AND "DB3500_UNIT_02_FIXTURE_1".UNCLAMPED_ANALOG;
END_REGION
END_FUNCTION
